FUNCTION Convert_LWORD_TO_BYTE : BOOL
VAR_INPUT
	in : LWORD;
	out : REFERENCE TO BYTE;
END_VAR
VAR
	converted : BYTE;
END_VAR

converted := LWORD_TO_BYTE(in);

IF (BYTE_TO_LWORD(converted) <> in) THEN
	RETURN;
END_IF

out := converted;
Convert_LWORD_TO_BYTE := TRUE;

END_FUNCTION

(* stored: Version 1.1.0.1, ProductVersion 3.1.4024.12
   POU Convert_LWORD_TO_BYTE: Id {bce4a70e-1a6b-42a1-8b58-65a52c8c18d5}, SpecialFunc None *)
